(* CODESYS project PowerDriveF300_MultiLeader.project

Project tree, tasks and I/O mapping:
  Powerdrive_Pump1 : Powerdrive F300, Nidec Control Techniques, version 1.10.9.2
    application Application
      Task Configuration
        Clock
      program Clock [ST]
      data type DataTimer
      data type DataRising
      data type DataOutput
      data type DataInput
      data type DataSet
      data type DataTemp
    RTEthernet
    SI_Ethernet : SI-Ethernet, Nidec Control Techniques, version 1.10.9.2
      RTEthernet
      Ethernet_1 : Ethernet, Nidec Control Techniques, version 1.10.9.2
    Ethernet : Ethernet, Nidec Control Techniques, version 1.10.9.2
    <Empty>
    <Empty>
  Powerdrive_Pump2 : Powerdrive F300, Nidec Control Techniques, version 1.10.9.2
    application Application
      data type DataOutput
      data type DataInput
      data type DataSet
      data type DataRising
      Task Configuration
        Clock
      program Clock [ST]
      data type DataTemp
      data type DataTimer
    RTEthernet
    SI_Ethernet : SI-Ethernet, Nidec Control Techniques, version 1.10.9.2
      RTEthernet
      Ethernet_1 : Ethernet, Nidec Control Techniques, version 1.10.9.2
    Ethernet : Ethernet, Nidec Control Techniques, version 1.10.9.2
    <Empty>
    <Empty>
  Powerdrive_Pump3 : Powerdrive F300, Nidec Control Techniques, version 1.10.9.2
    application Application
      Task Configuration
        Clock
      program Clock [ST]
      data type DataInput
      data type DataOutput
      data type DataRising
      data type DataSet
      data type DataTemp
      data type DataTimer
    RTEthernet
    Ethernet : Ethernet, Nidec Control Techniques, version 1.10.9.2
    <Empty>
    <Empty>
    SI_Ethernet : SI-Ethernet, Nidec Control Techniques, version 1.10.9.2
      RTEthernet
      Ethernet_1 : Ethernet, Nidec Control Techniques, version 1.10.9.2
  Advanced Link Editor
*)

// Powerdrive_Pump2/Application/DataOutput
TYPE DataOutput :
STRUCT
	o_Cycle :INT;
	o_RunAuto :BOOL;
	o_RunMan :BOOL;
END_STRUCT
END_TYPE

// Powerdrive_Pump2/Application/DataInput
TYPE DataInput :
STRUCT
	iAuto :BOOL;
	iReady :BOOL;
	iMan  :BOOL;
	hMan :BOOL;	
END_STRUCT
END_TYPE

// Powerdrive_Pump2/Application/DataSet
TYPE DataSet :
STRUCT
	FreqManual: INT;
	OutputFreq: INT;
	TimeCycle : INT;
	DelayCallPump: INT;
	DelayDisPump: INT;
END_STRUCT
END_TYPE

// Powerdrive_Pump2/Application/DataRising
TYPE DataRising :
STRUCT
	CLK_Auto :BOOL;
	Q_Auto :BOOL;
END_STRUCT
END_TYPE

// Powerdrive_Pump1/Application/DataTimer
TYPE DataTimer :
STRUCT
	InTimer :BOOL;
	PtTimer : TIME;
	PulseTimer : BOOL;
END_STRUCT
END_TYPE

// Powerdrive_Pump1/Application/DataRising
TYPE DataRising :
STRUCT
	CLK_Auto :BOOL;
	Q_Auto :BOOL;
END_STRUCT
END_TYPE

// Powerdrive_Pump1/Application/DataOutput
TYPE DataOutput :
STRUCT
	o_Cycle :INT;
	o_RunAuto :BOOL;
	o_RunMan :BOOL;
	runing :BOOL;
END_STRUCT
END_TYPE

// Powerdrive_Pump1/Application/DataInput
TYPE DataInput :
STRUCT
	iAuto :BOOL;
	iReady :BOOL;
	iMan  :BOOL;
	hMan :BOOL;	
END_STRUCT
END_TYPE

// Powerdrive_Pump1/Application/DataSet
TYPE DataSet :
	STRUCT		
	FreqManual: INT;
	OutputFreq: INT;
	TimeCycle : INT;
	DelayCallPump: INT;
	DelayDisPump: INT;
	END_STRUCT
END_TYPE

// Powerdrive_Pump1/Application/DataTemp
TYPE DataTemp :
STRUCT
	CountCycle : INT;
	CountCallPump :INT;
	Countdischarge :INT;
	t_AutoRun :BOOL;
	t_callPumpCycle :BOOL;
	t_CallPumpBooter: BOOL;
END_STRUCT
END_TYPE

// Powerdrive_Pump2/Application/DataTemp
TYPE DataTemp :
STRUCT
	CountCycle : INT;
	CountCallPump :INT;
	Countdischarge :INT;
	t_AutoRun :BOOL;
	t_callPumpCycle :BOOL;
	t_CallPumpBooter: BOOL;
END_STRUCT
END_TYPE

// Powerdrive_Pump2/Application/DataTimer
TYPE DataTimer :
STRUCT
	InTimer :BOOL;
	PtTimer : TIME;
	PulseTimer : BOOL;
END_STRUCT
END_TYPE

// Powerdrive_Pump3/Application/DataInput
TYPE DataInput :
	STRUCT
		iAuto :BOOL;
		iReady :BOOL;
		iMan  :BOOL;
		hMan :BOOL;	
	END_STRUCT
END_TYPE

// Powerdrive_Pump3/Application/DataOutput
TYPE DataOutput :
STRUCT
	o_Cycle :INT;
	o_RunAuto :BOOL;
	o_RunMan :BOOL;
END_STRUCT
END_TYPE

// Powerdrive_Pump3/Application/DataRising
TYPE DataRising :
STRUCT
	CLK_Auto :BOOL;
	Q_Auto :BOOL;
END_STRUCT
END_TYPE

// Powerdrive_Pump3/Application/DataSet
TYPE DataSet :
STRUCT
	FreqManual: INT;
	OutputFreq: INT;
	TimeCycle : INT;
	DelayCallPump: INT;
	DelayDisPump: INT;
END_STRUCT
END_TYPE

// Powerdrive_Pump3/Application/DataTemp
TYPE DataTemp :
STRUCT
	CountCycle : INT;
	CountCallPump :INT;
	Countdischarge :INT;
	t_AutoRun :BOOL;
	t_callPumpCycle :BOOL;
	t_CallPumpBooter: BOOL;
END_STRUCT
END_TYPE

// Powerdrive_Pump3/Application/DataTimer
TYPE DataTimer :
STRUCT
	InTimer :BOOL;
	PtTimer : TIME;
	PulseTimer : BOOL;
END_STRUCT
END_TYPE

// Powerdrive_Pump1/Application/Clock
PROGRAM Clock
VAR
	iPump1 :DataInput;
	oPump1 :DataOutput;
	iPump2 :DataInput;
	oPump2 :DataOutput;
	iPump3 :DataInput;
	oPump3 :DataOutput;
	
	AllAuto :DataRising;
	FirtCycle: R_TRIG;

	Timer1Second: TON;
	DataT1 : DataTimer;	
	temp_case:INT;	
	
	MasterSet :DataSet;
	TempOperation : DataTemp;
	t_Continue :BOOL;
	t_CallP1Man :BOOL;
END_VAR

// Program for Pump 1

// Run Manual with fixed frequency if ImanT23 and not Auto T24
iPump1.iMan := CTUniM.M08.P006;
iPump1.hMan := CTUniM.M19.P031;

iPump1.iAuto := CTUniM.M08.P003; // T24
iPump2.iAuto := CTUniM.M08.P004; // T25
iPump3.iAuto := CTUniM.M08.P005; // T26
iPump1.iReady := CTUniM.M10.P001;
MasterSet.FreqManual := CTUniM.M19.P011;
MasterSet.TimeCycle := CTUniM.M19.P012;
MasterSet.OutputFreq:= CTUniM.M19.P013;
MasterSet.DelayCallPump:= CTUniM.M19.P014;
MasterSet.DelayDisPump :=CTUniM.M19.P015;

IF CTUniM.M20.P008 =1 THEN
	iPump2.iReady := TRUE;
ELSE
	iPump2.iReady := FALSE;
END_IF
IF CTUniM.M20.P014 =1 THEN
	iPump3.iReady := TRUE;
ELSE
	iPump3.iReady := FALSE;
END_IF
// Check auto run case
IF  NOT iPump1.iMan AND iPump1.iAuto AND iPump2.iAuto AND iPump3.iAuto AND iPump1.iReady AND iPump2.iReady AND iPump3.iReady THEN  // All auto 1-2-3
	 temp_case:=1;	 
ELSE IF  NOT iPump1.iMan AND iPump1.iAuto AND iPump2.iAuto AND iPump1.iReady AND iPump2.iReady AND NOT iPump3.iAuto THEN   // 1-2 Auto
	temp_case:=2;
ELSE IF  NOT iPump1.iMan AND iPump1.iAuto AND NOT iPump2.iAuto AND iPump3.iAuto AND iPump1.iReady AND iPump3.iReady THEN   // 1-3 Auto
	temp_case:=3;
ELSE IF  NOT iPump1.iMan AND NOT iPump1.iAuto AND iPump2.iAuto AND iPump3.iAuto AND iPump2.iReady AND iPump3.iReady THEN   // 2-3 Auto
	temp_case:=4;
ELSE IF  NOT iPump1.iMan AND iPump1.iAuto AND NOT iPump2.iAuto AND NOT iPump3.iAuto THEN   // 1 Auto
	temp_case:=5;	
ELSE
	temp_case:=0;
END_IF
END_IF
END_IF
END_IF
END_IF
// 
	FirtCycle(CLK:=AllAuto.CLK_Auto , Q=>AllAuto.Q_Auto );
	DataT1.InTimer := NOT DataT1.PulseTimer;
	Timer1Second(IN:=DataT1.InTimer , PT:=T#1S , Q=>DataT1.PulseTimer , ET=> );
//
//
CASE temp_case OF
// Case 0  all auto	off
	0: 	TempOperation.CountCycle := 0;
		TempOperation.Countdischarge := 0;
		TempOperation.CountCallPump :=0;
		oPump1.o_RunAuto:=FALSE;
		oPump2.o_RunAuto:=FALSE;
		TempOperation.t_callPumpCycle :=FALSE;
		TempOperation.t_CallPumpBooter := FALSE;
// Case 1 Run Pump 1 Pump 2 and Pump 3
	1: 
		// Output temp runing pump		
		oPump1.o_RunAuto := iPump1.iAuto AND iPump1.iReady  AND NOT TempOperation.t_callPumpCycle ;
		oPump2.o_RunAuto := iPump2.iAuto AND iPump2.iReady AND NOT iPump2.iMan AND TempOperation.t_callPumpCycle;	
		oPump2.o_RunMan := iPump2.iAuto AND iPump2.iReady AND NOT TempOperation.t_callPumpCycle AND TempOperation.t_CallPumpBooter;
		
		oPump3.o_RunAuto := iPump3.iAuto AND iPump3.iReady AND NOT iPump3.iMan AND NOT iPump2.iReady AND TempOperation.t_callPumpCycle;
		oPump3.o_RunMan := iPump3.iAuto AND iPump2.iReady AND NOT iPump2.iReady AND NOT TempOperation.t_callPumpCycle AND TempOperation.t_CallPumpBooter;
		
		IF (oPump1.o_RunAuto AND NOT oPump2.o_RunAuto AND NOT oPump3.o_RunAuto) THEN
			oPump1.o_Cycle :=10;		
		ELSE IF ((NOT iPump1.iReady OR oPump2.o_RunAuto) AND iPump2.iReady) THEN
			oPump1.o_Cycle :=12;  // Transfer Master to pump 2	
		ELSE IF ((NOT iPump1.iReady OR oPump3.o_RunAuto) AND iPump3.iReady) THEN
			oPump1.o_Cycle :=13;  // Transfer Master to pump 3
		ELSE
			oPump1.o_Cycle :=0;
			END_IF
			END_IF
		END_IF
		
		// Time Cyle master PID
		IF(oPump1.o_RunAuto AND CTUniM.M10.P002 AND NOT TempOperation.t_callPumpCycle  AND DataT1.PulseTimer) THEN
			TempOperation.CountCycle := TempOperation.CountCycle +1;
		END_IF
		IF TempOperation.CountCycle >= MasterSet.TimeCycle THEN
			TempOperation.t_callPumpCycle :=TRUE;
			t_Continue :=TRUE;
			IF TempOperation.t_CallPumpBooter THEN
				TempOperation.t_CallPumpBooter := FALSE;
			END_IF			
		END_IF
		IF (t_Continue AND CTUniM.M20.P016=31) THEN
			TempOperation.t_callPumpCycle :=FALSE;
			t_Continue :=FALSE;
			TempOperation.CountCycle := 0;
		END_IF
		// Run PID and not enought pressure
		IF (CTUniM.M05.P001_RAW >= MasterSet.OutputFreq AND NOT TempOperation.t_CallPumpBooter AND NOT TempOperation.t_callPumpCycle AND DataT1.PulseTimer) THEN
			TempOperation.CountCallPump := TempOperation.CountCallPump +1;
			TempOperation.Countdischarge := 0;
		END_IF
		IF TempOperation.CountCallPump >= MasterSet.DelayCallPump THEN
			TempOperation.t_CallPumpBooter := TRUE;	
		END_IF
		// Runing booter and output frequenct decrease
		IF (TempOperation.t_CallPumpBooter AND CTUniM.M05.P001_RAW < MasterSet.OutputFreq) THEN
			TempOperation.Countdischarge := TempOperation.Countdischarge +1;
		END_IF
		IF TempOperation.Countdischarge  >= MasterSet.DelayDisPump THEN
			TempOperation.t_CallPumpBooter := FALSE;
			TempOperation.CountCallPump :=0;	
		END_IF
// Case 2 Run Pump 1 and Pump 2		
	2: 
		// Output temp runing pump		
		oPump1.o_RunAuto := iPump1.iAuto AND iPump1.iReady  AND NOT TempOperation.t_callPumpCycle ;
		oPump2.o_RunAuto := iPump2.iAuto AND iPump2.iReady AND NOT iPump2.iMan AND TempOperation.t_callPumpCycle;	
		oPump2.o_RunMan := iPump2.iAuto AND iPump2.iReady AND NOT TempOperation.t_callPumpCycle AND TempOperation.t_CallPumpBooter;
		IF (oPump1.o_RunAuto AND NOT oPump2.o_RunAuto) THEN
			oPump1.o_Cycle :=10;		
		ELSE IF ((NOT iPump1.iReady OR oPump2.o_RunAuto) AND iPump2.iReady) THEN
			oPump1.o_Cycle :=12;  // Transfer Master to pump 2		
		ELSE
			oPump1.o_Cycle :=0;
			END_IF
		END_IF
		// Time Cyle master PID
		IF(oPump1.o_RunAuto AND CTUniM.M10.P002 AND NOT TempOperation.t_callPumpCycle  AND DataT1.PulseTimer) THEN
			TempOperation.CountCycle := TempOperation.CountCycle +1;
		END_IF
		IF TempOperation.CountCycle >= MasterSet.TimeCycle THEN
			TempOperation.t_callPumpCycle :=TRUE;
			IF TempOperation.t_CallPumpBooter THEN
				TempOperation.t_CallPumpBooter := FALSE;
			END_IF			
		END_IF
		IF oPump2.o_RunAuto AND CTUniM.M20.P010=21 THEN
			TempOperation.t_callPumpCycle :=FALSE;
			TempOperation.CountCycle := 0;
		END_IF
		// Run PID and not enought pressure
		IF (CTUniM.M05.P001_RAW >= MasterSet.OutputFreq  AND NOT TempOperation.t_CallPumpBooter AND NOT TempOperation.t_callPumpCycle AND DataT1.PulseTimer) THEN
			TempOperation.CountCallPump := TempOperation.CountCallPump +1;
			TempOperation.Countdischarge := 0;
		END_IF
		IF TempOperation.CountCallPump >= MasterSet.DelayCallPump THEN
			TempOperation.t_CallPumpBooter := TRUE;	
		END_IF
		// Runing booter and output frequenct decrease
		IF (TempOperation.t_CallPumpBooter AND CTUniM.M05.P001_RAW < MasterSet.OutputFreq) THEN
			TempOperation.Countdischarge := TempOperation.Countdischarge +1;
		END_IF
		IF TempOperation.Countdischarge  >= MasterSet.DelayDisPump THEN
			TempOperation.t_CallPumpBooter := FALSE;
			TempOperation.CountCallPump :=0;	
		END_IF
// Case 1 Run Pump 1 and Pump 3
	3:
		// Output temp runing pump		
		oPump1.o_RunAuto := iPump1.iAuto AND iPump1.iReady  AND NOT TempOperation.t_callPumpCycle ;
		oPump3.o_RunAuto := iPump3.iAuto AND iPump3.iReady AND NOT iPump3.iMan AND TempOperation.t_callPumpCycle;	
		oPump3.o_RunMan := iPump3.iAuto AND iPump3.iReady AND NOT TempOperation.t_callPumpCycle AND TempOperation.t_CallPumpBooter;
		IF (oPump1.o_RunAuto AND NOT oPump3.o_RunAuto) THEN
			oPump1.o_Cycle :=10;		
		ELSE IF ((NOT iPump1.iReady OR oPump3.o_RunAuto) AND iPump3.iReady) THEN
			oPump1.o_Cycle :=13;  // Transfer Master to pump 3		
		ELSE
			oPump1.o_Cycle :=0;
			END_IF
		END_IF
		// Time Cyle master PID
		IF(oPump1.o_RunAuto AND CTUniM.M10.P002 AND NOT TempOperation.t_callPumpCycle  AND DataT1.PulseTimer) THEN
			TempOperation.CountCycle := TempOperation.CountCycle +1;
		END_IF
		IF TempOperation.CountCycle >= MasterSet.TimeCycle THEN
			TempOperation.t_callPumpCycle :=TRUE;
			IF TempOperation.t_CallPumpBooter THEN
				TempOperation.t_CallPumpBooter := FALSE;
			END_IF			
		END_IF
		IF oPump3.o_RunAuto AND CTUniM.M20.P016=31 THEN
			TempOperation.t_callPumpCycle :=FALSE;
			TempOperation.CountCycle := 0;
		END_IF
		// Run PID and not enought pressure
		IF (CTUniM.M05.P001_RAW >= MasterSet.OutputFreq  AND NOT TempOperation.t_CallPumpBooter AND NOT TempOperation.t_callPumpCycle AND DataT1.PulseTimer) THEN
			TempOperation.CountCallPump := TempOperation.CountCallPump +1;
			TempOperation.Countdischarge := 0;
		END_IF
		IF TempOperation.CountCallPump >= MasterSet.DelayCallPump THEN
			TempOperation.t_CallPumpBooter := TRUE;	
		END_IF
		// Runing booter and output frequenct decrease
		IF (TempOperation.t_CallPumpBooter AND CTUniM.M05.P001_RAW < MasterSet.OutputFreq) THEN
			TempOperation.Countdischarge := TempOperation.Countdischarge +1;
		END_IF
		IF TempOperation.Countdischarge  >= MasterSet.DelayDisPump THEN
			TempOperation.t_CallPumpBooter := FALSE;
			TempOperation.CountCallPump :=0;	
		END_IF
// Case 4 Run Pump 2 and Pump 3
	4:
		TempOperation.CountCycle := 0;
		TempOperation.Countdischarge := 0;
		TempOperation.CountCallPump :=0;
// Case 5 Run Pump 1
	5:	
		oPump1.o_RunAuto := iPump1.iAuto AND iPump1.iReady ;
	
END_CASE
// Runing command Manual and Auto
IF CTUniM.M20.P012=1 OR CTUniM.M20.P018=1 THEN
	t_CallP1Man:=TRUE;
ELSE
	t_CallP1Man:=FALSE;
END_IF
IF 	(iPump1.iMan OR iPump1.hMan OR t_CallP1Man)  THEN
	oPump1.o_Cycle :=14;
	CTUniM.M06.P034 := iPump1.iMan OR iPump1.hMan OR (t_CallP1Man AND iPump1.iAuto);
	CTUniM.M01.P021_RAW := MasterSet.FreqManual;
ELSE IF NOT iPump1.iMan AND iPump1.iAuto THEN
		CTUniM.M06.P034 := oPump1.o_RunAuto;
		CTUniM.M14.P008 :=oPump1.o_RunAuto;
		CTUniM.M01.P021_RAW :=CTUniM.M14.P001_RAW/10;
ELSE
	CTUniM.M06.P034 := FALSE;
	CTUniM.M14.P008 := FALSE;
	CTUniM.M01.P021_RAW := 0;
	oPump1.o_Cycle :=0;
	END_IF
END_IF
// Call Pump 2 compensation
IF oPump2.o_RunMan THEN
	CTUniM.M18.P013:= 2;  // call pump 2
ELSE IF oPump3.o_RunMan THEN
	CTUniM.M18.P013:= 3;   // call pump 3
ELSE
	CTUniM.M18.P013:= 0;
END_IF
END_IF
CTUniM.M08.P031 := oPump2.o_RunMan;
CTUniM.M08.P032 := oPump3.o_RunMan;
CTUniM.M19.P020 := TempOperation.CountCycle;
CTUniM.M19.P021 := TempOperation.CountCallPump;
CTUniM.M19.P022 := TempOperation.Countdischarge;
// Transfer infor to Pump 2
CTUniM.M18.P011 := oPump1.o_Cycle; 
IF  CTUniM.M18.P011 =14 THEN
	CTUniM.M18.P040 :=TRUE;
ELSE
	CTUniM.M18.P040 :=FALSE;
END_IF
IF  CTUniM.M18.P011 =10 THEN
	CTUniM.M18.P041 :=TRUE;
ELSE
	CTUniM.M18.P041 :=FALSE;
END_IF

END_PROGRAM

// Powerdrive_Pump2/Application/Clock
PROGRAM Clock
VAR
	iPump1 :DataInput;
	oPump1 :DataOutput;
	iPump2 :DataInput;
	oPump2 :DataOutput;
	iPump3 :DataInput;
	oPump3 :DataOutput;
	
	AllAuto :DataRising;
	FirtCycle: R_TRIG;

	Timer1Second: TON;
	DataT1 : DataTimer;	
	temp_case:INT;	
	
	MasterSet :DataSet;
	TempOperation : DataTemp;
	t_CallP2 :BOOL;
	t_CallP2Man :BOOL;
END_VAR

// Program for Pump 2

// Run Manual with fixed frequency if ImanT23 and not Auto T24
iPump1.iMan := CTUniM.M08.P006; // T27
iPump2.hMan := CTUniM.M19.P031;

iPump1.iAuto := CTUniM.M08.P003; // T24
iPump2.iAuto := CTUniM.M08.P004; // T25
iPump3.iAuto := CTUniM.M08.P005; // T26
iPump2.iReady := CTUniM.M10.P001;
MasterSet.FreqManual := CTUniM.M19.P011;
MasterSet.TimeCycle := CTUniM.M19.P012;
MasterSet.OutputFreq:= CTUniM.M19.P013;
MasterSet.DelayCallPump:= CTUniM.M19.P014;
MasterSet.DelayDisPump :=CTUniM.M19.P015;

IF CTUniM.M20.P002 =1 THEN
	iPump1.iReady := TRUE;
ELSE
	iPump1.iReady := FALSE;
END_IF
IF CTUniM.M20.P014 =1 THEN
	iPump3.iReady := TRUE;
ELSE
	iPump3.iReady := FALSE;
END_IF

// Check auto run case
IF  NOT iPump2.iMan AND iPump1.iAuto AND iPump2.iAuto AND iPump3.iAuto AND iPump1.iReady AND iPump2.iReady AND iPump3.iReady THEN  // All auto 1-2-3
	 temp_case:=1;	 
ELSE IF  NOT iPump2.iMan AND iPump1.iAuto AND iPump2.iAuto AND iPump1.iReady AND iPump2.iReady AND NOT iPump3.iAuto THEN   // 1-2 Auto
	temp_case:=2;
ELSE IF  NOT iPump2.iMan AND iPump1.iAuto AND NOT iPump2.iAuto AND iPump3.iAuto AND iPump1.iReady AND iPump3.iReady THEN   // 1-3 Auto
	temp_case:=3;
ELSE IF  NOT iPump2.iMan AND NOT iPump1.iAuto AND iPump2.iAuto AND iPump3.iAuto AND iPump2.iReady AND iPump3.iReady THEN   // 2-3 Auto
	temp_case:=4;	
ELSE IF  NOT iPump2.iMan AND iPump2.iAuto AND NOT iPump1.iAuto AND NOT iPump3.iAuto THEN   // 2-3 Auto
	temp_case:=5;
ELSE
	temp_case:=0;
END_IF
END_IF
END_IF
END_IF
END_IF
// 
	FirtCycle(CLK:=AllAuto.CLK_Auto , Q=>AllAuto.Q_Auto );
	DataT1.InTimer := NOT DataT1.PulseTimer;
	Timer1Second(IN:=DataT1.InTimer , PT:=T#1S , Q=>DataT1.PulseTimer , ET=> );
//
//
CASE temp_case OF
// Case 0 Off all auto	
	0: 	TempOperation.CountCycle := 0;
		TempOperation.Countdischarge := 0;
		TempOperation.CountCallPump :=0;
		oPump1.o_RunAuto:=FALSE;
		oPump2.o_RunAuto:=FALSE;
		TempOperation.t_callPumpCycle :=FALSE;
		TempOperation.t_CallPumpBooter := FALSE;
// Case 1 Run Pump 1 Pump 2 and Pump 3
	1: 
		// Output temp runing pump	
		IF (CTUniM.M20.P004 =12 OR CTUniM.M20.P016=32) THEN
			t_CallP2 := TRUE;
		END_IF	
		oPump2.o_RunAuto := iPump2.iAuto AND iPump2.iReady AND t_CallP2 AND NOT TempOperation.t_callPumpCycle ;
		oPump3.o_RunAuto := iPump3.iAuto AND iPump3.iReady AND NOT iPump3.iMan AND TempOperation.t_callPumpCycle;	
		oPump3.o_RunMan := iPump3.iAuto AND iPump3.iReady AND NOT TempOperation.t_callPumpCycle AND TempOperation.t_CallPumpBooter;
		
		oPump1.o_RunAuto := iPump1.iAuto AND iPump1.iReady AND NOT iPump1.iMan AND NOT iPump3.iReady AND TempOperation.t_callPumpCycle;
		oPump1.o_RunMan := iPump1.iAuto AND iPump1.iReady  AND NOT iPump3.iReady AND NOT TempOperation.t_callPumpCycle AND TempOperation.t_CallPumpBooter;
		IF (oPump2.o_RunAuto AND NOT oPump3.o_RunAuto AND NOT oPump1.o_RunAuto) THEN
			oPump2.o_Cycle :=20;		
		ELSE IF ((NOT iPump2.iReady OR oPump3.o_RunAuto) AND iPump3.iReady) THEN
			oPump2.o_Cycle :=23;  // Transfer Master to pump 3	
		ELSE IF ((NOT iPump1.iReady OR oPump1.o_RunAuto) AND iPump1.iReady) THEN
			oPump2.o_Cycle :=21;  // Transfer Master to pump 1		
		ELSE
			oPump2.o_Cycle :=0;
			END_IF
			END_IF
		END_IF
		// Time Cyle master PID
		IF(oPump2.o_RunAuto AND CTUniM.M10.P002 AND NOT TempOperation.t_callPumpCycle  AND DataT1.PulseTimer) THEN
			TempOperation.CountCycle := TempOperation.CountCycle +1;
		END_IF
		IF TempOperation.CountCycle >= MasterSet.TimeCycle THEN
			TempOperation.t_callPumpCycle :=TRUE;
			IF TempOperation.t_CallPumpBooter THEN
				TempOperation.t_CallPumpBooter := FALSE;
			END_IF			
		END_IF
		IF (t_CallP2 AND CTUniM.M20.P004=10) THEN
			TempOperation.t_callPumpCycle :=FALSE;
			t_CallP2 := FALSE;
			TempOperation.CountCycle := 0;
		END_IF
		// Run PID and not enought pressure
		IF (CTUniM.M05.P001_RAW >= MasterSet.OutputFreq AND NOT TempOperation.t_CallPumpBooter AND NOT TempOperation.t_callPumpCycle AND DataT1.PulseTimer) THEN
			TempOperation.CountCallPump := TempOperation.CountCallPump +1;
			TempOperation.Countdischarge := 0;
		END_IF
		IF TempOperation.CountCallPump >= MasterSet.DelayCallPump THEN
			TempOperation.t_CallPumpBooter := TRUE;	
		END_IF
		// Runing booter and output frequenct decrease
		IF (TempOperation.t_CallPumpBooter AND CTUniM.M05.P001_RAW < MasterSet.OutputFreq) THEN
			TempOperation.Countdischarge := TempOperation.Countdischarge +1;
		END_IF
		IF TempOperation.Countdischarge  >= MasterSet.DelayDisPump THEN
			TempOperation.t_CallPumpBooter := FALSE;
			TempOperation.CountCallPump :=0;	
		END_IF
// Case 2 Run Pump 1 and Pump 2		
	2: 
		// Output temp runing pump		
		oPump2.o_RunAuto := iPump2.iAuto AND iPump2.iReady AND CTUniM.M20.P004 =12 AND NOT TempOperation.t_callPumpCycle ;
		oPump1.o_RunAuto := iPump1.iAuto AND iPump1.iReady AND NOT iPump1.iMan AND TempOperation.t_callPumpCycle;	
		oPump1.o_RunMan := iPump1.iAuto AND iPump1.iReady AND NOT TempOperation.t_callPumpCycle AND TempOperation.t_CallPumpBooter;
		IF (oPump2.o_RunAuto AND NOT oPump2.o_RunAuto) THEN
			oPump2.o_Cycle :=20;		
		ELSE IF ((NOT iPump2.iReady OR oPump2.o_RunAuto) AND iPump1.iReady) THEN
			oPump2.o_Cycle :=21;  // Transfer Master to pump 1		
		ELSE
			oPump2.o_Cycle :=0;
			END_IF
		END_IF
		// Time Cyle master PID
		IF(oPump2.o_RunAuto AND CTUniM.M10.P002 AND NOT TempOperation.t_callPumpCycle  AND DataT1.PulseTimer) THEN
			TempOperation.CountCycle := TempOperation.CountCycle +1;
		END_IF
		IF TempOperation.CountCycle >= MasterSet.TimeCycle THEN
			TempOperation.t_callPumpCycle :=TRUE;
			IF TempOperation.t_CallPumpBooter THEN
				TempOperation.t_CallPumpBooter := FALSE;
			END_IF			
		END_IF
		IF oPump1.o_RunAuto AND CTUniM.M20.P004=12 THEN
			TempOperation.t_callPumpCycle :=FALSE;
			TempOperation.CountCycle := 0;
		END_IF
		// Run PID and not enought pressure
		IF (CTUniM.M05.P001_RAW >= MasterSet.OutputFreq  AND NOT TempOperation.t_CallPumpBooter AND NOT TempOperation.t_callPumpCycle AND DataT1.PulseTimer) THEN
			TempOperation.CountCallPump := TempOperation.CountCallPump +1;
			TempOperation.Countdischarge := 0;
		END_IF
		IF TempOperation.CountCallPump >= MasterSet.DelayCallPump THEN
			TempOperation.t_CallPumpBooter := TRUE;	
		END_IF
		// Runing booter and output frequenct decrease
		IF (TempOperation.t_CallPumpBooter AND CTUniM.M05.P001_RAW < MasterSet.OutputFreq) THEN
			TempOperation.Countdischarge := TempOperation.Countdischarge +1;
		END_IF
		IF TempOperation.Countdischarge  >= MasterSet.DelayDisPump THEN
			TempOperation.t_CallPumpBooter := FALSE;
			TempOperation.CountCallPump :=0;	
		END_IF
// Case 1 Run Pump 1 and Pump 3
	3:
		TempOperation.CountCycle := 0;
		TempOperation.Countdischarge := 0;
		TempOperation.CountCallPump :=0;
// Case 1 Run Pump 2 and Pump 3
	4:
		// Output temp runing pump		
		oPump2.o_RunAuto := iPump2.iAuto AND iPump2.iReady  AND NOT TempOperation.t_callPumpCycle ;
		oPump3.o_RunAuto := iPump3.iAuto AND iPump3.iReady AND NOT iPump3.iMan AND TempOperation.t_callPumpCycle;	
		oPump3.o_RunMan := iPump3.iAuto AND iPump3.iReady AND NOT TempOperation.t_callPumpCycle AND TempOperation.t_CallPumpBooter;
		IF (oPump2.o_RunAuto AND NOT oPump3.o_RunAuto ) THEN
			oPump2.o_Cycle :=20;		
		ELSE IF ((NOT iPump1.iReady OR oPump3.o_RunAuto) AND iPump3.iReady) THEN
			oPump2.o_Cycle :=23;  // Transfer Master to pump 3			
		ELSE
			oPump2.o_Cycle :=0;
			END_IF
		END_IF
		// Time Cyle master PID
		IF(oPump2.o_RunAuto AND CTUniM.M10.P002 AND NOT TempOperation.t_callPumpCycle  AND DataT1.PulseTimer) THEN
			TempOperation.CountCycle := TempOperation.CountCycle +1;
		END_IF
		IF TempOperation.CountCycle >= MasterSet.TimeCycle THEN
			TempOperation.t_callPumpCycle :=TRUE;
			IF TempOperation.t_CallPumpBooter THEN
				TempOperation.t_CallPumpBooter := FALSE;
				TempOperation.CountCallPump :=0;
				TempOperation.Countdischarge := 0;
			END_IF			
		END_IF
		IF oPump3.o_RunAuto AND CTUniM.M20.P016=32 THEN
			TempOperation.t_callPumpCycle :=FALSE;
			TempOperation.CountCycle := 0;
		END_IF
		// Run PID and not enought pressure
		IF (CTUniM.M05.P001_RAW >= MasterSet.OutputFreq AND NOT TempOperation.t_CallPumpBooter AND NOT TempOperation.t_callPumpCycle AND DataT1.PulseTimer) THEN
			TempOperation.CountCallPump := TempOperation.CountCallPump +1;
			TempOperation.Countdischarge := 0;
		END_IF
		IF TempOperation.CountCallPump >= MasterSet.DelayCallPump THEN
			TempOperation.t_CallPumpBooter := TRUE;	
		END_IF
		// Runing booter and output frequenct decrease
		IF (TempOperation.t_CallPumpBooter AND CTUniM.M05.P001_RAW < MasterSet.OutputFreq) THEN
			TempOperation.Countdischarge := TempOperation.Countdischarge +1;
		END_IF
		IF TempOperation.Countdischarge  >= MasterSet.DelayDisPump THEN
			TempOperation.t_CallPumpBooter := FALSE;
			TempOperation.CountCallPump :=0;	
		END_IF
// Case 5 Run Pump 2		
	5:
		oPump2.o_RunAuto := iPump2.iAuto AND iPump2.iReady ;
	
END_CASE
// Runing command Manual and Auto
IF CTUniM.M20.P006=2 OR CTUniM.M20.P018=2 THEN
	t_CallP2Man:=TRUE;
ELSE
	t_CallP2Man:=FALSE;
END_IF
IF 	(iPump2.iMan OR iPump2.hMan OR t_CallP2Man)  THEN
	oPump2.o_Cycle :=24;
	CTUniM.M06.P034 := iPump2.iMan OR iPump2.hMan OR (t_CallP2Man AND iPump2.iAuto) ;
	CTUniM.M01.P021_RAW := MasterSet.FreqManual;
ELSE IF NOT iPump2.iMan AND iPump2.iAuto THEN
		CTUniM.M06.P034 := oPump2.o_RunAuto;
		CTUniM.M14.P008 :=oPump2.o_RunAuto;
		CTUniM.M01.P021_RAW :=CTUniM.M14.P001_RAW/10;
ELSE
	CTUniM.M06.P034 := FALSE;
	CTUniM.M14.P008 := FALSE;
	CTUniM.M01.P021_RAW := 0;
	oPump2.o_Cycle :=0;
	END_IF
END_IF
// Call Pump 3 compensation
IF oPump3.o_RunMan THEN
	CTUniM.M18.P013:= 3; // call pump 3
ELSE IF oPump1.o_RunMan THEN
	CTUniM.M18.P013:= 1;   // call pump 1
ELSE
	CTUniM.M18.P013:= 0;
END_IF
END_IF

CTUniM.M08.P031 := oPump2.o_RunMan;
CTUniM.M08.P032 := oPump3.o_RunMan;
CTUniM.M19.P020 := TempOperation.CountCycle;
CTUniM.M19.P021 := TempOperation.CountCallPump;
CTUniM.M19.P022 := TempOperation.Countdischarge;
// Transfer infor to Pump 2
CTUniM.M18.P011 := oPump2.o_Cycle; 
IF  CTUniM.M18.P011 =24 THEN
	CTUniM.M18.P040 :=TRUE;
ELSE
	CTUniM.M18.P040 :=FALSE;
END_IF
IF  CTUniM.M18.P011 =20 THEN
	CTUniM.M18.P041 :=TRUE;
ELSE
	CTUniM.M18.P041 :=FALSE;
END_IF

END_PROGRAM

// Powerdrive_Pump3/Application/Clock
PROGRAM Clock
VAR
	iPump1 :DataInput;
	oPump1 :DataOutput;
	iPump2 :DataInput;
	oPump2 :DataOutput;
	iPump3 :DataInput;
	oPump3 :DataOutput;
	
	AllAuto :DataRising;
	FirtCycle: R_TRIG;

	Timer1Second: TON;
	DataT1 : DataTimer;	
	temp_case:INT;	
	
	MasterSet :DataSet;
	TempOperation : DataTemp;
	t_CallP3 :BOOL;
	t_CallP3Man :BOOL;
END_VAR

// Program for Pump 3

// Run Manual with fixed frequency if ImanT23 and not Auto T24
iPump1.iMan := CTUniM.M08.P006; // T27
iPump3.hMan := CTUniM.M19.P031;

iPump1.iAuto := CTUniM.M08.P003; // T24
iPump2.iAuto := CTUniM.M08.P004; // T25
iPump3.iAuto := CTUniM.M08.P005; // T26
iPump3.iReady := CTUniM.M10.P001;
MasterSet.FreqManual := CTUniM.M19.P011;
MasterSet.TimeCycle := CTUniM.M19.P012;
MasterSet.OutputFreq:= CTUniM.M19.P013;
MasterSet.DelayCallPump:= CTUniM.M19.P014;
MasterSet.DelayDisPump :=CTUniM.M19.P015;
IF CTUniM.M20.P002 =1 THEN
	iPump1.iReady := TRUE;
ELSE
	iPump1.iReady := FALSE;
END_IF
IF CTUniM.M20.P008 =1 THEN
	iPump2.iReady := TRUE;
ELSE
	iPump2.iReady := FALSE;
END_IF

// Check auto run case
IF  NOT iPump3.iMan AND iPump1.iAuto AND iPump2.iAuto AND iPump3.iAuto AND iPump1.iReady AND iPump2.iReady AND iPump3.iReady THEN  // All auto 1-2-3
	 temp_case:=1;	 
ELSE IF  NOT iPump3.iMan AND iPump1.iAuto AND iPump2.iAuto AND iPump1.iReady AND iPump2.iReady AND NOT iPump3.iAuto THEN   // 1-2 Auto
	temp_case:=2;
ELSE IF  NOT iPump3.iMan AND iPump1.iAuto AND NOT iPump2.iAuto AND iPump3.iAuto AND iPump1.iReady AND iPump3.iReady THEN   // 1-3 Auto
	temp_case:=3;
ELSE IF  NOT iPump3.iMan AND NOT iPump1.iAuto AND iPump2.iAuto AND iPump3.iAuto AND iPump2.iReady AND iPump3.iReady THEN   // 2-3 Auto
	temp_case:=4;	
ELSE IF  NOT iPump3.iMan AND iPump3.iAuto AND NOT iPump1.iAuto AND NOT iPump2.iAuto THEN   // 2-3 Auto
	temp_case:=5;	
ELSE
	temp_case:=0;
END_IF
END_IF
END_IF
END_IF
END_IF
// 
	FirtCycle(CLK:=AllAuto.CLK_Auto , Q=>AllAuto.Q_Auto );
	DataT1.InTimer := NOT DataT1.PulseTimer;
	Timer1Second(IN:=DataT1.InTimer , PT:=T#1S , Q=>DataT1.PulseTimer , ET=> );
//
//
CASE temp_case OF
// Off all auto	
	0: 	TempOperation.CountCycle := 0;
		TempOperation.Countdischarge := 0;
		TempOperation.CountCallPump :=0;
		oPump1.o_RunAuto:=FALSE;
		oPump2.o_RunAuto:=FALSE;
		TempOperation.t_callPumpCycle :=FALSE;
		TempOperation.t_CallPumpBooter := FALSE;
// Case 1 Run Pump 1 Pump 2 and Pump 3
	1: 
		// Output temp runing pump	
		IF (CTUniM.M20.P004 =13  OR CTUniM.M20.P010 =23 ) THEN
			t_CallP3 := TRUE;
		END_IF	
		oPump3.o_RunAuto := iPump3.iAuto AND iPump3.iReady AND t_CallP3 AND NOT TempOperation.t_callPumpCycle ;
		oPump1.o_RunAuto := iPump1.iAuto AND iPump1.iReady AND NOT iPump1.iMan AND TempOperation.t_callPumpCycle;	
		oPump1.o_RunMan := iPump1.iAuto AND iPump1.iReady AND NOT TempOperation.t_callPumpCycle AND TempOperation.t_CallPumpBooter;
		
		oPump2.o_RunAuto := iPump2.iAuto AND iPump2.iReady AND NOT iPump2.iMan AND NOT iPump1.iReady AND TempOperation.t_callPumpCycle;
		oPump2.o_RunMan := iPump2.iAuto AND iPump2.iReady AND NOT iPump1.iReady  AND NOT TempOperation.t_callPumpCycle AND TempOperation.t_CallPumpBooter;
		IF (oPump3.o_RunAuto AND NOT oPump1.o_RunAuto AND NOT oPump2.o_RunAuto) THEN
			oPump3.o_Cycle :=30;		
		ELSE IF ((NOT iPump3.iReady OR oPump1.o_RunAuto) AND iPump1.iReady) THEN
			oPump3.o_Cycle :=31;  // Transfer Master to pump 1		
		ELSE IF ((NOT iPump3.iReady OR oPump2.o_RunAuto) AND iPump2.iReady) THEN
			oPump3.o_Cycle :=32;  // Transfer Master to pump 2		
		ELSE
			oPump3.o_Cycle :=0;
			END_IF
			END_IF
		END_IF
		// Time Cyle master PID
		IF(oPump3.o_RunAuto AND CTUniM.M10.P002 AND NOT TempOperation.t_callPumpCycle  AND DataT1.PulseTimer) THEN
			TempOperation.CountCycle := TempOperation.CountCycle +1;
		END_IF
		IF TempOperation.CountCycle >= MasterSet.TimeCycle THEN
			TempOperation.t_callPumpCycle :=TRUE;
			IF TempOperation.t_CallPumpBooter THEN
				TempOperation.t_CallPumpBooter := FALSE;
			END_IF			
		END_IF
		IF (t_CallP3 AND CTUniM.M20.P004 =10) THEN
			TempOperation.t_callPumpCycle :=FALSE;
			t_CallP3 := FALSE;
			TempOperation.CountCycle := 0;
		END_IF
		// Run PID and not enought pressure
		IF (CTUniM.M05.P001_RAW >= MasterSet.OutputFreq AND NOT TempOperation.t_CallPumpBooter AND NOT TempOperation.t_callPumpCycle AND DataT1.PulseTimer) THEN
			TempOperation.CountCallPump := TempOperation.CountCallPump +1;
			TempOperation.Countdischarge := 0;
		END_IF
		IF TempOperation.CountCallPump >= MasterSet.DelayCallPump THEN
			TempOperation.t_CallPumpBooter := TRUE;	
		END_IF
		// Runing booter and output frequenct decrease
		IF (TempOperation.t_CallPumpBooter AND CTUniM.M05.P001_RAW < MasterSet.OutputFreq) THEN
			TempOperation.Countdischarge := TempOperation.Countdischarge +1;
		END_IF
		IF TempOperation.Countdischarge  >= MasterSet.DelayDisPump THEN
			TempOperation.t_CallPumpBooter := FALSE;
			TempOperation.CountCallPump :=0;	
		END_IF
// Case 2 Run Pump 1 and Pump 2		
	2: 
		TempOperation.CountCycle := 0;
		TempOperation.Countdischarge := 0;
		TempOperation.CountCallPump :=0;
// Case 1 Run Pump 1 and Pump 3
	3:
		// Output temp runing pump		
		oPump3.o_RunAuto := iPump3.iAuto AND iPump3.iReady AND CTUniM.M20.P004 =13  AND NOT TempOperation.t_callPumpCycle ;
		oPump1.o_RunAuto := iPump1.iAuto AND iPump1.iReady AND NOT iPump1.iMan AND TempOperation.t_callPumpCycle;	
		oPump1.o_RunMan := iPump1.iAuto AND iPump1.iReady AND NOT TempOperation.t_callPumpCycle AND TempOperation.t_CallPumpBooter;
		IF (oPump3.o_RunAuto AND NOT oPump3.o_RunAuto) THEN
			oPump3.o_Cycle :=30;		
		ELSE IF ((NOT iPump3.iReady OR oPump1.o_RunAuto) AND iPump1.iReady) THEN
			oPump3.o_Cycle :=31;  // Transfer Master to pump 1		
		ELSE
			oPump3.o_Cycle :=0;
			END_IF
		END_IF
		// Time Cyle master PID
		IF(oPump3.o_RunAuto AND CTUniM.M10.P002 AND NOT TempOperation.t_callPumpCycle  AND DataT1.PulseTimer) THEN
			TempOperation.CountCycle := TempOperation.CountCycle +1;
		END_IF
		IF TempOperation.CountCycle >= MasterSet.TimeCycle THEN
			TempOperation.t_callPumpCycle :=TRUE;
			IF TempOperation.t_CallPumpBooter THEN
				TempOperation.t_CallPumpBooter := FALSE;
			END_IF			
		END_IF
		IF oPump1.o_RunAuto AND CTUniM.M20.P004 =13 THEN
			TempOperation.t_callPumpCycle :=FALSE;
			TempOperation.CountCycle := 0;
		END_IF
		// Run PID and not enought pressure
		IF (CTUniM.M05.P001_RAW >= MasterSet.OutputFreq  AND NOT TempOperation.t_CallPumpBooter AND NOT TempOperation.t_callPumpCycle AND DataT1.PulseTimer) THEN
			TempOperation.CountCallPump := TempOperation.CountCallPump +1;
			TempOperation.Countdischarge := 0;
		END_IF
		IF TempOperation.CountCallPump >= MasterSet.DelayCallPump THEN
			TempOperation.t_CallPumpBooter := TRUE;	
		END_IF
		// Runing booter and output frequenct decrease
		IF (TempOperation.t_CallPumpBooter AND CTUniM.M05.P001_RAW < MasterSet.OutputFreq) THEN
			TempOperation.Countdischarge := TempOperation.Countdischarge +1;
		END_IF
		IF TempOperation.Countdischarge  >= MasterSet.DelayDisPump THEN
			TempOperation.t_CallPumpBooter := FALSE;
			TempOperation.CountCallPump :=0;	
		END_IF
// Case 1 Run Pump 2 and Pump 3
	4:
		// Output temp runing pump		
		oPump3.o_RunAuto := iPump3.iAuto AND iPump3.iReady AND CTUniM.M20.P010 =23 AND NOT TempOperation.t_callPumpCycle ;
		oPump2.o_RunAuto := iPump2.iAuto AND iPump2.iReady AND NOT iPump2.iMan AND TempOperation.t_callPumpCycle;	
		oPump2.o_RunMan := iPump2.iAuto AND iPump2.iReady AND NOT TempOperation.t_callPumpCycle AND TempOperation.t_CallPumpBooter;
		IF (oPump3.o_RunAuto AND NOT oPump2.o_RunAuto) THEN
			oPump3.o_Cycle :=30;		
		ELSE IF ((NOT iPump3.iReady OR oPump2.o_RunAuto) AND iPump2.iReady) THEN
			oPump3.o_Cycle :=32;  // Transfer Master to pump 3			
		ELSE
			oPump3.o_Cycle :=0;
			END_IF
		END_IF
		// Time Cyle master PID
		IF(oPump3.o_RunAuto AND CTUniM.M10.P002 AND NOT TempOperation.t_callPumpCycle  AND DataT1.PulseTimer) THEN
			TempOperation.CountCycle := TempOperation.CountCycle +1;
		END_IF
		IF TempOperation.CountCycle >= MasterSet.TimeCycle THEN
			TempOperation.t_callPumpCycle :=TRUE;
			IF TempOperation.t_CallPumpBooter THEN
				TempOperation.t_CallPumpBooter := FALSE;
			END_IF			
		END_IF
		IF oPump2.o_RunAuto AND CTUniM.M20.P010 =23 THEN
			TempOperation.t_callPumpCycle :=FALSE;
			TempOperation.CountCycle := 0;
			TempOperation.CountCallPump :=0;
			TempOperation.Countdischarge := 0;
		END_IF
		// Run PID and not enought pressure
		IF (CTUniM.M05.P001_RAW >= MasterSet.OutputFreq  AND NOT TempOperation.t_CallPumpBooter AND NOT TempOperation.t_callPumpCycle AND DataT1.PulseTimer) THEN
			TempOperation.CountCallPump := TempOperation.CountCallPump +1;
			TempOperation.Countdischarge := 0;
		END_IF
		IF TempOperation.CountCallPump >= MasterSet.DelayCallPump THEN
			TempOperation.t_CallPumpBooter := TRUE;	
		END_IF
		// Runing booter and output frequenct decrease
		IF (TempOperation.t_CallPumpBooter AND CTUniM.M05.P001_RAW < MasterSet.OutputFreq) THEN
			TempOperation.Countdischarge := TempOperation.Countdischarge +1;
		END_IF
		IF TempOperation.Countdischarge  >= MasterSet.DelayDisPump THEN
			TempOperation.t_CallPumpBooter := FALSE;
			TempOperation.CountCallPump :=0;	
		END_IF
// Case 5 Run Pump 2		
	5:
		oPump3.o_RunAuto := iPump3.iAuto AND iPump3.iReady ;
	
END_CASE
// Runing command Manual and Auto
IF CTUniM.M20.P006=3 OR CTUniM.M20.P012=3 THEN
	t_CallP3Man:=TRUE;
ELSE
	t_CallP3Man:=FALSE;
END_IF
IF 	(iPump3.iMan OR iPump3.hMan OR t_CallP3Man)  THEN
	oPump3.o_Cycle :=34;
	CTUniM.M06.P034 := iPump3.iMan OR iPump3.hMan OR (t_CallP3Man AND iPump3.iAuto) ;
	CTUniM.M01.P021_RAW := MasterSet.FreqManual;
ELSE IF NOT iPump3.iMan AND iPump3.iAuto THEN
		CTUniM.M06.P034 := oPump3.o_RunAuto;
		CTUniM.M14.P008 :=oPump3.o_RunAuto;
		CTUniM.M01.P021_RAW :=CTUniM.M14.P001_RAW/10;
ELSE
	CTUniM.M06.P034 := FALSE;
	CTUniM.M14.P008 := FALSE;
	CTUniM.M01.P021_RAW := 0;
	oPump3.o_Cycle :=0;
	END_IF
END_IF
// Call Pump 2 compensation
IF oPump2.o_RunMan THEN
	CTUniM.M18.P013:= 2; // call pump 2
ELSE IF oPump1.o_RunMan THEN
	CTUniM.M18.P013:= 1; // call pump 1
ELSE
	CTUniM.M18.P013:= 0;
END_IF
END_IF
CTUniM.M08.P031 := oPump2.o_RunMan;
CTUniM.M08.P032 := oPump3.o_RunMan;
CTUniM.M19.P020 := TempOperation.CountCycle;
CTUniM.M19.P021 := TempOperation.CountCallPump;
CTUniM.M19.P022 := TempOperation.Countdischarge;
// Transfer infor to Pump 2
CTUniM.M18.P011 := oPump3.o_Cycle;
IF  CTUniM.M18.P011 =34 THEN
	CTUniM.M18.P040 :=TRUE;
ELSE
	CTUniM.M18.P040 :=FALSE;
END_IF
IF  CTUniM.M18.P011 =30 THEN
	CTUniM.M18.P041 :=TRUE;
ELSE
	CTUniM.M18.P041 :=FALSE;
END_IF

END_PROGRAM
